TYPE "PLCtoMES_AGVExchange"
VERSION : 0.1
   STRUCT
      "P-MaterielCall" : Byte;
      "P-PosCall1" : Byte;
      "P-PosCall2" : Byte;
      "P-PosCall3" : Byte;
      "P-PosCall4" : Byte;
      "P-PosCall5" : Byte;
      "P-PalletNo1" : String[38];
      "P-PalletNo2" : String[38];
      "P-PalletNo3" : String[38];
      "P-PalletNo4" : String[38];
      "P-PalletNo5" : String[38];
      Reserve : Array[1..794] of Byte;
   END_STRUCT;

END_TYPE

